FUNCTION TryConvert_USINT_TO_UDINT : BOOL
VAR_INPUT
	in : USINT;
	out : REFERENCE TO UDINT;
END_VAR

out := USINT_TO_UDINT(in);
TryConvert_USINT_TO_UDINT := TRUE;

END_FUNCTION

(* stored: Version 1.1.0.1, ProductVersion 3.1.4024.12
   POU TryConvert_USINT_TO_UDINT: Id {c5807844-547d-4b67-991a-d2307f9f8062}, SpecialFunc None *)
